// TwinCAT 3 PLC project Libraries
// Title: Logging/file library
// Company: Ziga
// Author: Ziga
// ProjectVersion: 0.0.1.1
// Description: A library containing file/logging functionalities.
// ProgramVersion: 3.1.4024.0
// libraries:
//   Tc2_Standard, * (Beckhoff Automation GmbH)
//   Tc2_System, * (Beckhoff Automation GmbH)
//   Tc2_Utilities, * (Beckhoff Automation GmbH)
//   Tc3_Module, * (Beckhoff Automation GmbH)
//   TcUnit, * (www.tcunit.org)
//   Core, * (Ziga)
// project tree:
//   SOURCE/01_FileHandling/DUTs/ E_FileOpenMode.TcDUT
//   SOURCE/01_FileHandling/POUs/ FB_FileHandler.TcPOU, I_FileHandler.TcIO (not stored)
//   SOURCE/02_Logging/DUTs/ E_LoggerState.TcDUT (not stored)
//   SOURCE/02_Logging/POUs/ FB_Logger.TcPOU (not stored)
//   / TestsTask.TcTTO (not stored)
//   TESTS/ PRG_TESTS.TcPOU (not stored)
//   TESTS/Test suites/ FB_FileHandler_Tests.TcPOU
//   Version/ Global_Version.TcGVL
// (motion and I/O tree: see PLC project io)
// real-time tasks:
//   TASK TestsTask: cycle T#10ms, priority 20, ADS port 350

// ---- SOURCE/01_FileHandling/DUTs/E_FileOpenMode.TcDUT
// A combination of file open modes, based on available options.
// Source: https://infosys.beckhoff.com/english.php?content=../content/1033/tcplclib_tc2_system/30977547.html&id=


TYPE E_FileOpenMode :
(
	(* r: Opens a file for reading. An error is returned if the file cannot be found or does not exist.*)
	TEXT_READ := Tc2_System.FOPEN_MODEREAD OR Tc2_System.FOPEN_MODETEXT,
	
	(* 	w: Opens an empty file for writing. If the file already exists, it is overwritten.*)
	TEXT_WRITE := Tc2_System.FOPEN_MODEWRITE OR Tc2_System.FOPEN_MODETEXT,
	
	(* a: Opens a file for writing at the end of the file (append). If the file does not exist, a new file is created.*)
	TEXT_APPEND := Tc2_System.FOPEN_MODEAPPEND OR Tc2_System.FOPEN_MODETEXT,
	
	(* r+: Opens a file for reading and writing. The file must exist.*)
	TEXT_READ_MUST_EXIST := Tc2_System.FOPEN_MODEREAD OR Tc2_System.FOPEN_MODEPLUS OR Tc2_System.FOPEN_MODETEXT,
	
	(* w+: Opens an empty file for reading and writing. If the file already exists, it is overwritten.*)
	TEXT_READ_WRITE_OVERWRITE_EXISTING := Tc2_System.FOPEN_MODEWRITE OR Tc2_System.FOPEN_MODEPLUS OR Tc2_System.FOPEN_MODETEXT,
	
	(* a+: opens a file for reading and writing at the end of the file (append). 
	If the file does not exist, a new file is created. For this, the memory path must be known, otherwise error 1804 appears. 
	All write operations are always performed at end of a file, if the file was opened in the modes a or a+.
	The file pointer can be moved with FB_FileSeek, although for writing it is moved to the end of the file by default, i.e. existing data cannot be overwritten.*)
	TEXT_READ_APPEND_OVERWRITE_EXISTING	:= Tc2_System.FOPEN_MODEAPPEND OR Tc2_System.FOPEN_MODEPLUS OR Tc2_System.FOPEN_MODETEXT,
	
	(* r: Opens a file for reading. An error is returned if the file cannot be found or does not exist.*)
	BINARY_READ	:= Tc2_System.FOPEN_MODEREAD OR Tc2_System.FOPEN_MODEBINARY,
	
	(* 	w: Opens an empty file for writing. If the file already exists, it is overwritten.*)
	BINARY_WRITE := Tc2_System.FOPEN_MODEWRITE OR Tc2_System.FOPEN_MODEBINARY,
	
	(* a: Opens a file for writing at the end of the file (append). If the file does not exist, a new file is created.*)
	BINARY_APPEND := Tc2_System.FOPEN_MODEAPPEND OR Tc2_System.FOPEN_MODEBINARY,
	
	(* r+: Opens a file for reading and writing. The file must exist.*)
	BINARY_READ_MUST_EXIST := Tc2_System.FOPEN_MODEREAD OR Tc2_System.FOPEN_MODEPLUS OR Tc2_System.FOPEN_MODEBINARY,
	
	(* w+: Opens an empty file for reading and writing. If the file already exists, it is overwritten.*)
	BINARY_READ_WRITE_OVERWRITE_EXISTING := Tc2_System.FOPEN_MODEWRITE OR Tc2_System.FOPEN_MODEPLUS OR Tc2_System.FOPEN_MODEBINARY,
	
	(* a+: opens a file for reading and writing at the end of the file (append). 
	If the file does not exist, a new file is created. For this, the memory path must be known, otherwise error 1804 appears. 
	All write operations are always performed at end of a file, if the file was opened in the modes a or a+.
	The file pointer can be moved with FB_FileSeek, although for writing it is moved to the end of the file by default, i.e. existing data cannot be overwritten.*)
	BINARY_READ_APPEND_OVERWRITE_EXISTING := Tc2_System.FOPEN_MODEAPPEND OR Tc2_System.FOPEN_MODEPLUS OR Tc2_System.FOPEN_MODEBINARY
)DWORD;
END_TYPE

// ---- Version/Global_Version.TcGVL
{attribute 'TcGenerated'}
{attribute 'no-analysis'}
{attribute 'linkalways'}
// This function has been automatically generated from the project information.
VAR_GLOBAL CONSTANT
	{attribute 'const_non_replaced'}
	stLibVersion_Logging_file_library : ST_LibVersion := (iMajor := 0, iMinor := 0, iBuild := 1, iRevision := 1, nFlags := 0, sVersion := '0.0.1.1');
END_VAR

// ---- SOURCE/01_FileHandling/POUs/FB_FileHandler.TcPOU
// A function block containing multiple file handling methods.
// For examples refer to tests in the folder "TESTS/Test suites", file "FB_FileHandlerTests".
FUNCTION_BLOCK FB_FileHandler IMPLEMENTS I_FileHandler

VAR
	_fileHandle		: UINT;
	_fileProperties	: ZigasLibs_Core.ST_FileProperties;
	_error			: BOOL;
	_amsAddress		: Tc2_System.ST_AmsAddr;
END_VAR

(* Gets or sets the Ams address structure*)
PROPERTY AmsAddress : REFERENCE TO ZigasLibs_Core.Tc2_System.ST_AmsAddr
GET
AmsAddress ref= _amsAddress;
END_GET
SET
_amsAddress := AmsAddress;
END_SET
END_PROPERTY

(* Closes the file (if opened). Returns TRUE when done - method needs to be called until it returns TRUE!*)
METHOD PRIVATE Close : BOOL

VAR_INST
	fbFileClose			: Tc2_System.FB_FileClose;
	nCloseFileState		: UINT;
END_VAR

VAR CONSTANT
	FILE_CLOSE_START 		: UINT := 0;
	FILE_CLOSE_WAIT_BUSY	: UINT := 10;
	FILE_CLOSE_DONE			: UINT := 20;
END_VAR
IF THIS^.HandleCreated = FALSE THEN
	Close := TRUE;
	RETURN;
END_IF

_error := _error OR fbFileClose.bError;

CASE nCloseFileState OF
	FILE_CLOSE_START:
		fbFileClose(bExecute := FALSE);
		fbFileClose(bExecute := TRUE, hFile := _fileHandle);
		nCloseFileState := FILE_CLOSE_WAIT_BUSY;
		
	FILE_CLOSE_WAIT_BUSY:
		fbFileClose(bExecute := FALSE);
		IF NOT fbFileClose.bBusy AND NOT fbFileClose.bError THEN
			nCloseFileState := FILE_CLOSE_DONE;
		END_IF

	FILE_CLOSE_DONE:
		Close := TRUE;
		_fileHandle := 0;
		nCloseFileState := FILE_CLOSE_START;
END_CASE
END_METHOD

(* Creates the file. Returns TRUE when done - method needs to be called until it returns TRUE!*)
METHOD Create : BOOL
VAR_INPUT
	(* If file already exists, it will be deleted and crated once again (content will be lost!)*)
	bOverwrite	: BOOL;
END_VAR

VAR_INST
	fbFileOpen	: Tc2_System.FB_FileOpen;
	nFileCreateState	: UINT;
END_VAR

VAR CONSTANT
	FILE_CREATE_STATE_START					: UINT := 0;
	FILE_CREATE_STATE_OVERWRITE_OR_CREATE	: UINT := 10;
	FILE_CREATE_STATE_WAIT_DONE				: UINT := 20;
	FILE_CREATE_STATE_DONE					: UINT := 30;
END_VAR
CASE nFileCreateState OF
	FILE_CREATE_STATE_START:
		nFileCreateState := FILE_CREATE_STATE_OVERWRITE_OR_CREATE;
		
	FILE_CREATE_STATE_OVERWRITE_OR_CREATE:
		IF bOverwrite THEN
			IF THIS^.Open(mode := E_FileOpenMode.BINARY_READ_WRITE_OVERWRITE_EXISTING) THEN
				nFileCreateState := FILE_CREATE_STATE_WAIT_DONE;
			END_IF
		ELSE
			IF THIS^.Open(mode := E_FileOpenMode.BINARY_APPEND) THEN
				nFileCreateState := FILE_CREATE_STATE_WAIT_DONE;
			END_IF
		END_IF
		
	FILE_CREATE_STATE_WAIT_DONE:
	IF THIS^.Close() THEN
		nFileCreateState := FILE_CREATE_STATE_DONE;
	END_IF

		
	FILE_CREATE_STATE_DONE:
		Create := TRUE;
		nFileCreateState := FILE_CREATE_STATE_START;
END_CASE
END_METHOD

(* Deletes the file, if it exists. Returns TRUE when done - method needs to be called until it returns TRUE!*)
METHOD Delete : BOOL

VAR_INST
	fbFileDelete		: Tc2_System.FB_FileDelete;
	FtrigDeleteFinished	: Tc2_Standard.F_TRIG;
	bCheckIfFileExists	: BOOL;
	bFileExists			: BOOL;
END_VAR
fbFileDelete(
	bExecute := NOT fbFileDelete.bBusy,
	sPathName := ZigasLibs_Core.FileHelper.CreateFilePath(_fileProperties.FileLocation, _fileProperties.FileName,  ''));
	
FtrigDeleteFinished(CLK := fbFileDelete.bBusy);
IF FtrigDeleteFinished.Q THEN
	fbFileDelete(bExecute := FALSE);
	Delete := TRUE;
END_IF

_error := _error OR fbFileDelete.bError;
END_METHOD

(* Gets the error state, if any of the functions failed.*)
PROPERTY Error : BOOL
GET
Error := _error;
END_GET
END_PROPERTY

(* Checks if the file exists. Returns TRUE when done - method needs to be called until it returns TRUE!*)
METHOD Exists : BOOL
VAR_INPUT
	(* When mehod is finished, the variable provided here will have the result, TRUE if file exists, FALSE if not.*)
	refFileExists	: REFERENCE TO BOOL;
END_VAR

VAR_INST
	fbFileExists			: Tc2_Utilities.FB_EnumFindFileEntry := (tTimeout := T#5S);
	nCheckFileExistState	: UINT;
END_VAR

VAR CONSTANT
	FILE_EXIST_STATE_PREPARE	: UINT := 0;
	FILE_EXIST_STATE_START		: UINT := 10;
	FILE_EXIST_STATE_CHECK		: UINT := 20;
	FILE_EXIST_STATE_DONE		: UINT := 30;
END_VAR
CASE nCheckFileExistState OF
	FILE_EXIST_STATE_PREPARE:
		fbFileExists(bExecute := FALSE, eCmd := Tc2_Utilities.E_EnumCmdType.eEnumCmd_First);
		refFileExists := FALSE;
		nCheckFileExistState := FILE_EXIST_STATE_START;
		
	FILE_EXIST_STATE_START:
		fbFileExists(bExecute := TRUE,
			sPathName := ZigasLibs_Core.FileHelper.CreateFilePath(_fileProperties.FileLocation, _fileProperties.FileName, ''),
			sNetId := ZigasLibs_Core.AmsHelper.NetIdToString(_amsAddress.netId));
		nCheckFileExistState := FILE_EXIST_STATE_CHECK;
	
	FILE_EXIST_STATE_CHECK:
		fbFileExists(bExecute := FALSE);
		IF NOT fbFileExists.bBusy THEN
			IF NOT fbFileExists.bError THEN
				IF fbFileExists.stFindFile.sFileName = _fileProperties.FileName THEN
					refFileExists := TRUE;
					nCheckFileExistState := FILE_EXIST_STATE_DONE;
				END_IF	
				IF NOT fbFileExists.bEOE THEN
					fbFileExists.eCmd := Tc2_Utilities.E_EnumCmdType.eEnumCmd_Next;
				ELSE
					refFileExists := FALSE;
					nCheckFileExistState := FILE_EXIST_STATE_DONE;
				END_IF
			ELSE
				nCheckFileExistState := FILE_EXIST_STATE_DONE;
				refFileExists := FALSE;
				_error := _error OR fbFileExists.bError;
			END_IF
		END_IF
	
	FILE_EXIST_STATE_DONE:
		Exists := TRUE;
		nCheckFileExistState := FILE_EXIST_STATE_PREPARE;
END_CASE
END_METHOD

(* Gets or sets various file properties*)
PROPERTY FileProperties : REFERENCE TO ZigasLibs_Core.ST_FileProperties
GET
FileProperties ref= _fileProperties;
END_GET
SET
_fileProperties := FileProperties;
END_SET
END_PROPERTY

(* Gets the state of the file handle - if file is opened and handle is created returns TRUE.*)
PROPERTY PRIVATE HandleCreated : BOOL
GET
HandleCreated := _fileHandle <> 0;
END_GET
END_PROPERTY

(* Opens the file. Returns TRUE when done - method needs to be called until it returns TRUE!*)
METHOD PRIVATE Open : BOOL
VAR_INPUT
	mode	: E_FileOpenMode;	// Mode in which the file is opened
END_VAR

VAR_INST
	fbFileOpen	: Tc2_System.FB_FileOpen;
END_VAR
IF THIS^.HandleCreated THEN
	Open := TRUE;
	_error := _error OR fbFileOpen.bError;
	RETURN;
END_IF

fbFileOpen(
	bExecute := NOT fbFileOpen.bBusy,
	sPathName := ZigasLibs_Core.FileHelper.CreateFilePath(_fileProperties.FileLocation, _fileProperties.FileName, ''),
	sNetId :=  ZigasLibs_Core.AmsHelper.NetIdToString(_amsAddress.netId),
	nMode := mode,
	hFile => _fileHandle);
END_METHOD

(* Reads the content of the opened file to the target buffer.
 Returns TRUE when done - method needs to be called until it returns TRUE!*)
METHOD Read : BOOL
VAR_INPUT
	(* Pointer to the buffer, where the file content will be read to.*)
	ptrBuffer	: PVOID;
	(* Size of the buffer - SIZEOF()*)
	nBufferSize	: UDINT;
END_VAR


VAR_INST
	fbFileRead	: Tc2_System.FB_FileRead;
	nReadState	: UINT;
END_VAR

VAR CONSTANT
	READ_STATE_OPEN		: UINT := 0;
	READ_STATE_START	: UINT := 10;
	READ_STATE_WAIT		: UINT := 20;
	READ_STATE_DONE		: UINT := 30;
END_VAR
// An error is triggered if handle is not created or buffer pointer is invalid
IF ptrBuffer = 0 OR nBufferSize = 0 THEN
	_error := TRUE;
	Read := TRUE;
	RETURN;
END_IF

CASE nReadState OF
	READ_STATE_OPEN:
		IF THIS^.Open(mode := E_FileOpenMode.BINARY_READ) THEN
			nReadState := READ_STATE_START;
		END_IF	

	READ_STATE_START:
		fbFileRead(bExecute := FALSE);
		fbFileRead(
			bExecute := TRUE,
			hFile := _fileHandle,
			pReadBuff := ptrBuffer,
			cbReadLen := nBufferSize);
			
		nReadState := READ_STATE_WAIT;
		
	READ_STATE_WAIT:
		fbFileRead(bExecute := FALSE);
		IF fbFileRead.bBusy = FALSE THEN
			IF THIS^.Close() THEN
				nReadState := READ_STATE_DONE;
			END_IF
		END_IF	

	READ_STATE_DONE:
		_error := _error OR fbFileRead.bError;
		Read := TRUE;
		nReadState := READ_STATE_OPEN;
		
END_CASE
END_METHOD

METHOD PRIVATE WriteBinary : BOOL
VAR_INPUT
	ptrSource	: POINTER TO BYTE;	// Pointer to the source to be written - use ADR().
	nSize		: UDINT;	// Size of the source variable - use SIZEOF().
	mode		: E_FileOpenMode;
END_VAR

VAR_INST
	fbFileWrite	: Tc2_System.FB_FileWrite;
	nWriteState	: UINT;
END_VAR

VAR CONSTANT
	WRITE_OPEN_FILE	: UINT := 0;
	WRITE_START 	: UINT := 10;
	WRITE_WAIT_DONE	: UINT := 20;
	WRITE_DONE		: UINT := 30;
END_VAR
CASE nWriteState OF
	WRITE_OPEN_FILE:
		IF THIS^.Open(mode := mode) THEN
			nWriteState := WRITE_START;
		END_IF

	WRITE_START:
		fbFileWrite(bExecute := FALSE);
		fbFileWrite(
			bExecute := TRUE,
			hFile := _fileHandle,
			pWriteBuff := ptrSource,
			cbWriteLen := nSize);
			
		nWriteState := WRITE_WAIT_DONE;
	
	WRITE_WAIT_DONE:
		fbFileWrite(bExecute := FALSE);
		IF NOT fbFileWrite.bBusy THEN
			IF THIS^.Close() THEN
				nWriteState := WRITE_DONE;
			END_IF
		END_IF 
	
	WRITE_DONE:
		WriteBinary := TRUE;
END_CASE
END_METHOD

// Writes the content to the end of the file (appends).
// Returns TRUE when done - method needs to be called until it returns TRUE!
METHOD WriteBinary_Append : BOOL
VAR_INPUT
	ptrSource	: POINTER TO BYTE;	// Pointer to the source to be written - use ADR().
	nSize		: UDINT;	// Size of the source variable - use SIZEOF().
END_VAR
WriteBinary_Append := THIS^.WriteBinary(
	nSize := nSize, 
	ptrSource := ptrSource, 
	mode := E_FileOpenMode.BINARY_APPEND);
END_METHOD

(* Writes the content to the the file (overwrites any existing content).
 Returns TRUE when done - method needs to be called until it returns TRUE!*)
METHOD WriteBinary_Overwrite : BOOL
VAR_INPUT
	(* Pointer to the source to be written - use ADR().*)
	ptrSource	: POINTER TO BYTE;
	(* Size of the source variable - use SIZEOF().*)
	nSize	: UDINT;
END_VAR
WriteBinary_Overwrite := THIS^.WriteBinary(
	nSize := nSize, 
	ptrSource := ptrSource, 
	mode := E_FileOpenMode.BINARY_READ_WRITE_OVERWRITE_EXISTING);
END_METHOD

METHOD PRIVATE WriteLine : BOOL
VAR_INPUT
	(* Text to be written.*)
	sContent	: Tc2_System.T_MaxString;
	mode		: E_FileOpenMode;
END_VAR

VAR_INST
	fbFilePuts		: Tc2_System.FB_FilePuts;
	nWriteLineState	: UINT;
END_VAR

VAR CONSTANT
	WRITE_LINE_STATE_OPEN	: UINT := 0;
	WRITE_LINE_STATE_WRITE	: UINT := 10;
	WRITE_LINE_STATE_CLOSE	: UINT := 20;
	WRITE_LINE_STATE_DONE	: UINT := 30;
END_VAR
CASE nWriteLineState OF
	WRITE_LINE_STATE_OPEN:
		IF THIS^.Open(mode := mode) THEN
			nWriteLineState := WRITE_LINE_STATE_WRITE;
			fbFilePuts(bExecute := FALSE);
			fbFilePuts(
				bExecute := TRUE,
				hFile := _fileHandle,
				sLine := sContent,
				sNetId := ZigasLibs_Core.AmsHelper.NetIdToString(_amsAddress.netId),
				tTimeout := T#2S);
		END_IF
	
	WRITE_LINE_STATE_WRITE:
		fbFilePuts(bExecute := FALSE);
		IF fbFilePuts.bBusy = FALSE THEN
			nWriteLineState := WRITE_LINE_STATE_CLOSE;
		END_IF
	
	WRITE_LINE_STATE_CLOSE:
		IF THIS^.Close() THEN
			nWriteLineState := WRITE_LINE_STATE_DONE;
		END_IF
	
	WRITE_LINE_STATE_DONE:
		WriteLine := TRUE;
END_CASE

_error := _error OR fbFilePuts.bError;
END_METHOD

// Writes the string content to the end of the file (appends). If the file does not exist, it will be created.
// Returns TRUE when done - method needs to be called until it returns TRUE!
METHOD WriteLine_Append : BOOL
VAR_INPUT
	(* Text to be written.*)
	sContent	: Tc2_System.T_MaxString;
END_VAR
WriteLine_Append := THIS^.WriteLine(
	sContent := sContent, 
	mode := E_FileOpenMode.TEXT_APPEND);
END_METHOD

(* Writes the string content to file and overwrites any existing content. If the file does not exist, it will be created.
 Returns TRUE when done - method needs to be called until it returns TRUE!*)
METHOD WriteLine_Overwrite : BOOL
VAR_INPUT
	(* Text to be written.*)
	sContent	: Tc2_System.T_MaxString;
END_VAR
WriteLine_Overwrite := THIS^.WriteLine(
	sContent := sContent,
	mode := E_FileOpenMode.TEXT_APPEND);
END_METHOD

END_FUNCTION_BLOCK

// ---- TESTS/Test suites/FB_FileHandler_Tests.TcPOU
// Subject under test
FUNCTION_BLOCK FB_FileHandler_Tests EXTENDS FB_TestSuite

// Create instance variables that will be accesible for all tests
VAR
	_fileHandler			: FB_FileHandler;
	_writeFileLineState		: (WRITE, CHECK_WRITE_ERROR, WRITE_DONE);
	_readFileState			: (CLEAR_PREVIOUS_RESULT, READ, READ_DONE);
	_deleteFileState		: (DELETE, CHECK_FILE_EXIST, DELETE_DONE);
	_existFileState			: (EXIST_CREATE, EXIST_CHECK, EXIST_DELETE, EXIST_DONE);
	_writeFileBytesState	: (WRITEBYTES_START, WRITEBYTES_WAIT, WRITEBYTES_CHECK_CONTENT, WRITEBYTES_DELETE, WRITEBYTES_DONE);
END_VAR

VAR CONSTANT
	FOLDER_PATH 				: Tc2_System.T_MaxString := 'C:\Work\GitHub\TwinCAT\ZigaCAT\Tests\FileHandler';
	FILE_NAME					: Tc2_System.T_MaxString := 'FileName.txt';
	TEST_FILE_CONTENT_TEXT 		: Tc2_System.T_MaxString := 'This is a test file content!';
	TEST_FILE_CONTENT_BINARY	: STRING(300) := 'In a world full of possibilities, every moment is a chance to embrace growth, explore new horizons, and ignite your inner potential. Believe in the power of change, stay curious, and never stop learning. Your journey is unique, and every step forward brings you closer to your dreams.';
END_VAR

// Call your test methods here
_fileHandler.FileProperties.FileLocation := FOLDER_PATH;
_fileHandler.FileProperties.FileName := FILE_NAME;

Test_01_WriteLineAppend_ExpectNoError();
Test_02_ReadFileContent();
Test_03_DeleteFile_ExpectFileNotExist();
Test_04_CheckFileDoesNotExist_WriteToFile_ExpectFileExist_Delete();
Test_05_WriteBinaryAppend_NewFile_ExpectSameContent();

METHOD PRIVATE Test_01_WriteLineAppend_ExpectNoError
VAR_INPUT
END_VAR

VAR_INST
	delay	: Tc2_Standard.TON;
END_VAR
TcUnit.TEST('Test_01_WriteLineAppend_ExpectNoError');

CASE _writeFileLineState OF
	WRITE:
		IF _fileHandler.WriteLine_Append(sContent := TEST_FILE_CONTENT_TEXT) THEN
			_writeFileLineState := CHECK_WRITE_ERROR;
			delay(IN := FALSE);
		END_IF

	CHECK_WRITE_ERROR:
		AssertFalse(Condition := _fileHandler.Error, Message := 'Writing to file cause an unexpected error!');
		_writeFileLineState := WRITE_DONE;
		
	WRITE_DONE:
		TcUnit.TEST_FINISHED();
	
END_CASE
END_METHOD

METHOD PRIVATE Test_02_ReadFileContent
VAR_INPUT
END_VAR

VAR_INST
	sFileReadContentResult	: Tc2_System.T_MaxString;
END_VAR
TcUnit.TEST('Test_02_ReadFileContent');

CASE _readFileState OF
	CLEAR_PREVIOUS_RESULT:
		sFileReadContentResult := '';
		_readFileState := READ;

	READ:
		IF _writeFileLineState = WRITE_DONE THEN
			IF _fileHandler.Read(
					nBufferSize := SIZEOF(sFileReadContentResult), 
					ptrBuffer := ADR(sFileReadContentResult)) 
			THEN
				AssertEquals_STRING(
					Expected := TEST_FILE_CONTENT_TEXT,
					Actual := sFileReadContentResult,
					Message := 'Reading content from file failed - content differs!');
			
				AssertFalse(
					Condition := _fileHandler.Error, 
					Message := 'Reading file content triggered an unexpected error!');
					
				_readFileState := READ_DONE;
			END_IF
		END_IF

	READ_DONE:
		TcUnit.TEST_FINISHED();
	
END_CASE
END_METHOD

METHOD PRIVATE Test_03_DeleteFile_ExpectFileNotExist
var
	bFileExist	: BOOL;
END_VAR
TcUnit.TEST('Test_03_DeleteFile_ExpectFileNotExist');

CASE _deleteFileState OF
	DELETE:
		IF _readFileState = READ_DONE THEN
			IF _fileHandler.Delete() THEN
				_deleteFileState := CHECK_FILE_EXIST;
			END_IF
		END_IF
	
	CHECK_FILE_EXIST:
		IF _fileHandler.Exists(refFileExists := bFileExist) THEN
			AssertFalse(Condition := bFileExist, Message := 'Deleting file failed - file still exists!');
			_deleteFileState := DELETE_DONE;
		END_IF
	
	DELETE_DONE:
		TcUnit.TEST_FINISHED();
END_CASE
END_METHOD

METHOD PRIVATE Test_04_CheckFileDoesNotExist_WriteToFile_ExpectFileExist_Delete
VAR_INPUT
END_VAR

VAR_INST
	bFileExists	: BOOL;
END_VAR
TcUnit.TEST('Test_04_CheckFileDoesNotExist_WriteToFile_ExpectFileExist_Delete');

CASE _existFileState OF
	EXIST_CREATE:
		IF _deleteFileState = DELETE_DONE THEN
			IF _fileHandler.Create(FALSE) THEN
				AssertFalse(Condition := _fileHandler.Error, Message := 'An unexpected error occured while creating a file!');
				_existFileState := EXIST_CHECK;
			END_IF
		END_IF
	
	EXIST_CHECK:
		IF _fileHandler.Exists(refFileExists := bFileExists) THEN
			AssertTrue(Condition := bFileExists, Message := 'Creating file failed! File was not found!');
			_existFileState := EXIST_DELETE;
		END_IF
		
	EXIST_DELETE:
		IF _fileHandler.Delete() THEN
			_existFileState := EXIST_DONE;
		END_IF
	
	EXIST_DONE:
		TcUnit.TEST_FINISHED();
END_CASE
END_METHOD

METHOD PRIVATE Test_05_WriteBinaryAppend_NewFile_ExpectSameContent
VAR_INPUT
END_VAR

VAR_INST
	sReadResult		: STRING(300);
	sExpectedResult	: STRING(300) := TEST_FILE_CONTENT_BINARY;
END_VAR
TcUnit.TEST('Test_05_WriteBinaryAppend_NewFile_ExpectSameContent');

CASE _writeFileBytesState OF
	WRITEBYTES_START:
		sReadResult := '';
		IF _existFileState = EXIST_DONE THEN
			_writeFileBytesState := WRITEBYTES_WAIT;
		END_IF
		
	WRITEBYTES_WAIT:
		IF _fileHandler.WriteBinary_Append(nSize := SIZEOF(TEST_FILE_CONTENT_BINARY), ptrSource := ADR(TEST_FILE_CONTENT_BINARY)) THEN
			AssertFalse(Condition := _fileHandler.Error, Message := 'An unexpected error occured while writing bytes to a file!');
			_writeFileBytesState := WRITEBYTES_CHECK_CONTENT;
		END_IF
	
	WRITEBYTES_CHECK_CONTENT:
		IF _fileHandler.Read(nBufferSize := SIZEOF(sReadResult), ptrBuffer := ADR(sReadResult)) THEN
			AssertEquals(Expected := sExpectedResult, Actual := sReadResult, Message := 'Writing multiple bytes to a file failed!');
			_writeFileBytesState := WRITEBYTES_DELETE;
		END_IF
	
	WRITEBYTES_DELETE:
		IF _fileHandler.Delete() THEN
			_writeFileBytesState := WRITEBYTES_DONE;
		END_IF
	
	WRITEBYTES_DONE:
		TcUnit.TEST_FINISHED();
		
END_CASE
END_METHOD

END_FUNCTION_BLOCK
